// Mitsubishi GX Works2 project: 타이머응용   PLC: Q02/Q02H

PROGRAM MAIN
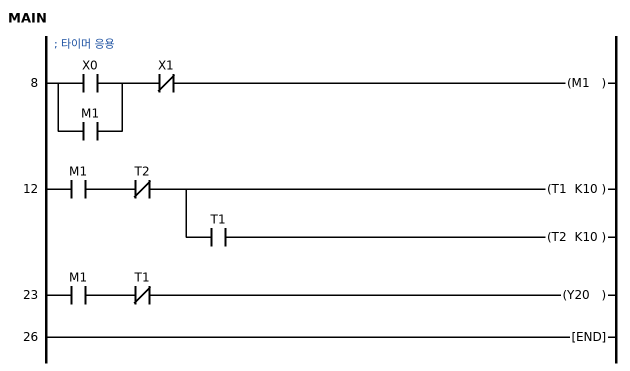
; 타이머 응용
8     LD      X0
      OR      M1
      ANI     X1
      OUT     M1
12    LD      M1
      ANI     T2
      OUT     T1 K10
      AND     T1
      OUT     T2 K10
23    LD      M1
      ANI     T1
      OUT     Y20
26    END
END_PROGRAM
